PROGRAM MAIN

END_PROGRAM

(* stored: Version 1.1.0.1
   POU MAIN: Id {faf4d8f6-3def-4c90-8920-6eff34c6bfa5}, SpecialFunc None *)
